// TIA Portal project "Tanques Mezcla Quimica" (V18)
// Llenado de tanques para mezcla quimica y tanque de almacenamiento

(* hardware
DEVICE "S7-1200 station_2"  S7-1200 Station
   slot 0: "Rack_0"  S7-1200 Rack  Rack  V1.0
   slot 1: "PLC_1"  CPU 1212C AC/DC/Rly  6ES7 212-1BE40-0XB0  V4.6
*)

// ===== PLC "PLC_1"  CPU 1212C AC/DC/Rly =====

VAR_GLOBAL   // PLC tag table "Default tag table_1"
   "Tag_1" AT %M1.4 : Bool;
END_VAR

VAR_GLOBAL CONSTANT   // PLC tag table "Default tag table_1"
   "None(1)" : Pip := 65535;
   "Automatic update(1)" : Pip := 0;
   "PIP 1(1)" : Pip := 1;
   "PIP 2(1)" : Pip := 2;
   "PIP 3(1)" : Pip := 3;
   "PIP 4(1)" : Pip := 4;
   "PIP OB Servo(1)" : Pip := 32768;
   "Local~MC(1)" : Hw_SubModule := 51;
   "Local~Common(1)" : Hw_SubModule := 50;
   "Local~Device(1)" : Hw_Device := 32;
   "Local~Configuration(1)" : Hw_SubModule := 33;
   "Local~Exec(1)" : Hw_SubModule := 52;
   "Local(1)" : Hw_SubModule := 49;
   "Local~PROFINET_interface_1(1)" : Hw_Interface := 64;
   "Local~PROFINET_interface_1~Port_1(1)" : Hw_Interface := 65;
   "Local~HSC_1(1)" : Hw_Hsc := 257;
   "Local~HSC_2(1)" : Hw_Hsc := 258;
   "Local~HSC_3(1)" : Hw_Hsc := 259;
   "Local~HSC_4(1)" : Hw_Hsc := 260;
   "Local~HSC_5(1)" : Hw_Hsc := 261;
   "Local~HSC_6(1)" : Hw_Hsc := 262;
   "Local~AI_2_1(1)" : Hw_SubModule := 263;
   "Local~DI_8_DQ_6_1(1)" : Hw_SubModule := 264;
   "Local~OPC_UA(1)" : Hw_SubModule := 117;
   "Local~Pulse_1(1)" : Hw_Pwm := 265;
   "Local~Pulse_2(1)" : Hw_Pwm := 266;
   "Local~Pulse_3(1)" : Hw_Pwm := 267;
   "Local~Pulse_4(1)" : Hw_Pwm := 268;
   "OB_Main(1)" : OB_PCYCLE := 1;
END_VAR

VAR_GLOBAL   // PLC tag table "IN"
   "START_MIX_PROCESS" AT %M0.0 : Bool;   // START PROCESS FOR MIX CHEMICHAL RECIPE
   "STOP_PROCESS" AT %M0.1 : Bool;   // STOP ALL THE PROCESS
   "EMERGENCY_STOP" AT %M0.2 : Bool;   // EMERGENCY STOP ALL THE PROCESS
   "TEMPERATURE_CONTROLLER" AT %M0.3 : Bool;   // TEMPERATURE CONTROLLER TANK C - CONTACT NO
   "LOW_LEVEL_TANK_C" AT %M0.4 : Bool;   // LOW LEVEL SENSOR TANK C - NO
   "LOW_LEVEL_TANK_A" AT %M0.5 : Bool;   // LOW LEVEL SENSOR TANK A - NO
   "LOW_LEVEL_TANK_B" AT %M0.6 : Bool;   // LOW LEVEL SENSOR TANK B - NO
   "HIGH_LEVEL_TANK_D" AT %M0.7 : Bool;   // HIGH LEVEL SENSOR TANK D - NO
END_VAR

VAR_GLOBAL   // PLC tag table "OUT"
   "VALVE_VA" AT %Q0.0 : Bool;   // ACTIVE VALVE A
   "VALVE_VB" AT %Q0.1 : Bool;   // ACTIVE VALVE B
   "VALVE_VD" AT %Q0.2 : Bool;   // ACTIVE VALVE D
   "PUMP" AT %Q0.3 : Bool;   // ACTIVE PUMP
   "HEATER_TANK_C" AT %Q0.4 : Bool;   // HEATER TANK C
   "VALVE_VC" AT %Q0.5 : Bool;   // ACTIVE VALVE C
END_VAR

// folder: GLOBAL VARIABLES

DATA_BLOCK "OUTPUTS"   // DB6
{ S7_Optimized_Access := 'TRUE' }
VERSION : 0.1
   VAR
      SET_RESET_PROCESS : Bool;   // START - STOP PROCESS
      OUT_TIMER_HEATER : Bool;   // OUTPUT TIMER HEATER
      OUT_TIMER_RESET_PROCESS : Bool;   // OUTPUT TIMER FOR RESET ALL PROCESS AUTO
   END_VAR
BEGIN
END_DATA_BLOCK

// folder: System blocks/Program resources

DATA_BLOCK "TIMER_DOSIFICATION_VALVE_A"   // DB1
{ S7_Optimized_Access := 'TRUE' }
AUTHOR : Simatic
FAMILY : IEC
NAME : IEC_TMR
VERSION : 1.0
// stored: InstanceOfName IEC_TIMER
"IEC_TIMER"
BEGIN
END_DATA_BLOCK

DATA_BLOCK "TIMER_DOSIFICATION_VALVE_B"   // DB2
{ S7_Optimized_Access := 'TRUE' }
AUTHOR : Simatic
FAMILY : IEC
NAME : IEC_TMR
VERSION : 1.0
// stored: InstanceOfName IEC_TIMER
"IEC_TIMER"
BEGIN
END_DATA_BLOCK

DATA_BLOCK "TIMER_HEATER_TANK_C"   // DB5
{ S7_Optimized_Access := 'TRUE' }
AUTHOR : Simatic
FAMILY : IEC
NAME : IEC_TMR
VERSION : 1.0
// stored: InstanceOfName IEC_TIMER
"IEC_TIMER"
BEGIN
END_DATA_BLOCK

DATA_BLOCK "TIMER_RESET_PROCESS"   // DB7
{ S7_Optimized_Access := 'TRUE' }
AUTHOR : Simatic
FAMILY : IEC
NAME : IEC_TMR
VERSION : 1.0
// stored: InstanceOfName IEC_TIMER
"IEC_TIMER"
BEGIN
END_DATA_BLOCK

// folder: TIMERS VALVE A-B

DATA_BLOCK "TIMERS_IN_OUT"   // DB3
{ S7_Optimized_Access := 'TRUE' }
VERSION : 0.1
   VAR
      OUT_TIMER_VA : Bool;   // OUTPUT TIMER VALVE A
      OUT_TIMER_VB : Bool;   // OUTPUT TIMER VALVE B
   END_VAR
BEGIN
END_DATA_BLOCK

// folder: (top level)

FUNCTION "START_STOP_PROCESS" : Void   // FC1, LAD
TITLE = SET - RESET PROCESS
{ S7_Optimized_Access := 'TRUE' }
VERSION : 0.1
// SET PROCESS
BEGIN

REGION Network 1: START PROCESS
   // SET PROCESS
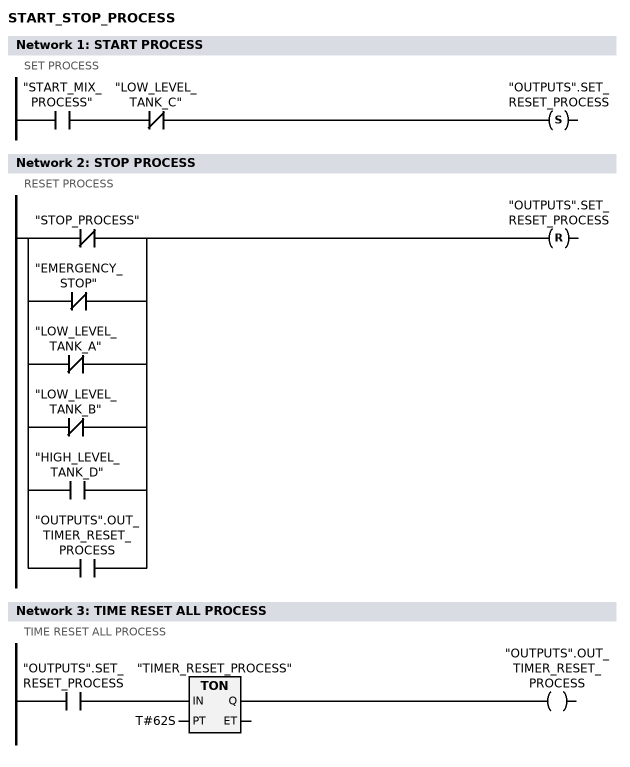
   RUNG wire#powerrail
      Contact( "START_MIX_PROCESS" )
      I_Contact( "LOW_LEVEL_TANK_C" )
      S_Coil( "OUTPUTS".SET_RESET_PROCESS )
   END_RUNG
   // the same network as SCL:
   IF "START_MIX_PROCESS" AND NOT "LOW_LEVEL_TANK_C" THEN "OUTPUTS".SET_RESET_PROCESS := TRUE; END_IF;
END_REGION

REGION Network 2: STOP PROCESS
   // RESET PROCESS
   RUNG wire#powerrail
      I_Contact( "STOP_PROCESS" )
      wire#w1
      R_Coil( "OUTPUTS".SET_RESET_PROCESS )
   END_RUNG
   RUNG wire#powerrail
      I_Contact( "EMERGENCY_STOP" )
   END_RUNG wire#w1
   RUNG wire#powerrail
      I_Contact( "LOW_LEVEL_TANK_A" )
   END_RUNG wire#w1
   RUNG wire#powerrail
      I_Contact( "LOW_LEVEL_TANK_B" )
   END_RUNG wire#w1
   RUNG wire#powerrail
      Contact( "HIGH_LEVEL_TANK_D" )
   END_RUNG wire#w1
   RUNG wire#powerrail
      Contact( "OUTPUTS".OUT_TIMER_RESET_PROCESS )
   END_RUNG wire#w1
   // the same network as SCL:
   IF NOT "STOP_PROCESS" OR NOT "EMERGENCY_STOP" OR NOT "LOW_LEVEL_TANK_A" OR NOT "LOW_LEVEL_TANK_B" OR "HIGH_LEVEL_TANK_D" OR "OUTPUTS".OUT_TIMER_RESET_PROCESS THEN
       "OUTPUTS".SET_RESET_PROCESS := FALSE;
   END_IF;
END_REGION

REGION Network 3: TIME RESET ALL PROCESS
   // TIME RESET ALL PROCESS
   "TIMER_RESET_PROCESS".TON(IN := "OUTPUTS".SET_RESET_PROCESS, PT := T#62S);
   "OUTPUTS".OUT_TIMER_RESET_PROCESS := "TIMER_RESET_PROCESS".Q;
END_REGION
END_FUNCTION

ORGANIZATION_BLOCK "Main"   // OB1, LAD, ProgramCycle
TITLE = "Main Program Sweep (Cycle)"
{ S7_Optimized_Access := 'TRUE' }
VERSION : 0.1
   VAR_INPUT
      Initial_Call : Bool;   // Initial call of this OB
      Remanence : Bool;   // =True, if remanent data are available
   END_VAR
BEGIN
END_ORGANIZATION_BLOCK

ORGANIZATION_BLOCK "Main_1"   // OB123, LAD, ProgramCycle
TITLE = "Main Program Sweep (Cycle)"
{ S7_Optimized_Access := 'TRUE' }
VERSION : 0.1
// ALL PROGRAM BLOCKS
   VAR_INPUT
      Initial_Call : Bool;   // Initial call of this OB
      Remanence : Bool;   // =True, if remanent data are available
   END_VAR
BEGIN

REGION Network 1: BLOCK SET - RESET PROCESS
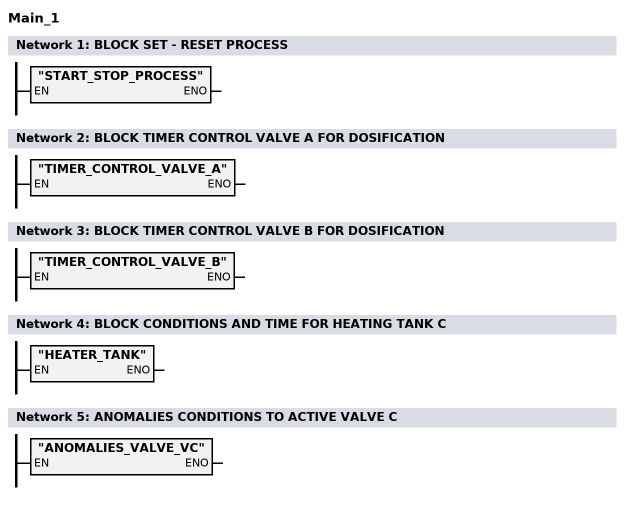
   RUNG wire#powerrail
      "START_STOP_PROCESS"()
   END_RUNG
   // the same network as SCL:
   "START_STOP_PROCESS"();
END_REGION

REGION Network 2: BLOCK TIMER CONTROL VALVE A FOR DOSIFICATION
   RUNG wire#powerrail
      "TIMER_CONTROL_VALVE_A"()
   END_RUNG
   // the same network as SCL:
   "TIMER_CONTROL_VALVE_A"();
END_REGION

REGION Network 3: BLOCK TIMER CONTROL VALVE B FOR DOSIFICATION
   RUNG wire#powerrail
      "TIMER_CONTROL_VALVE_B"()
   END_RUNG
   // the same network as SCL:
   "TIMER_CONTROL_VALVE_B"();
END_REGION

REGION Network 4: BLOCK CONDITIONS AND TIME FOR HEATING TANK C
   RUNG wire#powerrail
      "HEATER_TANK"()
   END_RUNG
   // the same network as SCL:
   "HEATER_TANK"();
END_REGION

REGION Network 5: ANOMALIES CONDITIONS TO ACTIVE VALVE C
   RUNG wire#powerrail
      "ANOMALIES_VALVE_VC"()
   END_RUNG
   // the same network as SCL:
   "ANOMALIES_VALVE_VC"();
END_REGION
END_ORGANIZATION_BLOCK

// folder: ANOMALIES CONDITIONS

FUNCTION "ANOMALIES_VALVE_VC" : Void   // FC5, LAD
TITLE = ANOMALIES TO ACTIVE VALVE C
{ S7_Optimized_Access := 'TRUE' }
VERSION : 0.1
// ANOMALIES CONDITIONS TO ACTIVE VALVE FOR DISCHARGE TANK C
BEGIN

REGION Network 1: ACTIVE VALVE C
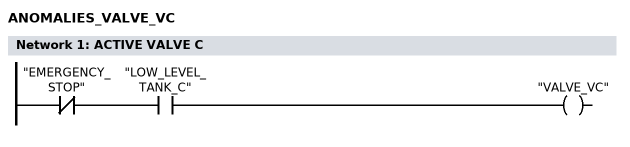
   RUNG wire#powerrail
      I_Contact( "EMERGENCY_STOP" )
      Contact( "LOW_LEVEL_TANK_C" )
      Coil( "VALVE_VC" )
   END_RUNG
   // the same network as SCL:
   "VALVE_VC" := NOT "EMERGENCY_STOP" AND "LOW_LEVEL_TANK_C";
END_REGION
END_FUNCTION

// folder: HEATER TANK C

FUNCTION "HEATER_TANK" : Void   // FC2, LAD
TITLE = START - STOP PROCESS OF HEATING, ACTIVE VALVE D AND PUMP
{ S7_Optimized_Access := 'TRUE' }
VERSION : 0.1
// CONDITIONS TO ACTIVE HEATER TANK C, CONDITIONS TO SET - RESET PUMP AND VALVE D
BEGIN

REGION Network 1: HEATER TANK C
   // CONDITIONS TO HEATING TANK C
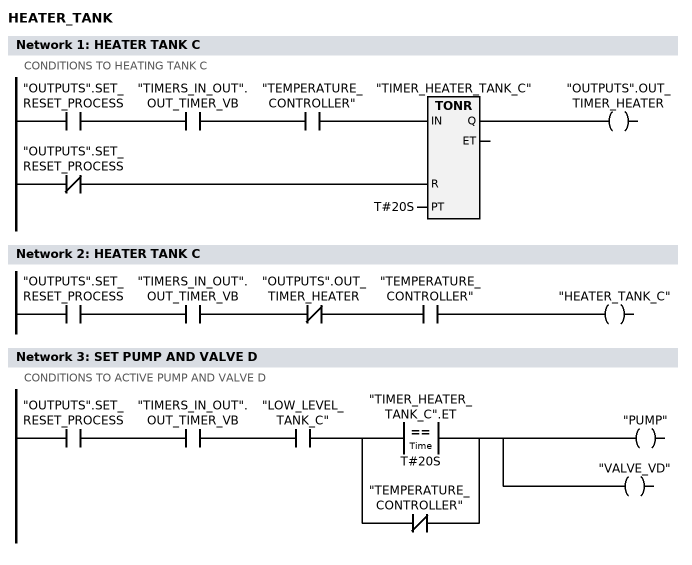
   "TIMER_HEATER_TANK_C".TONR(IN := "OUTPUTS".SET_RESET_PROCESS AND "TIMERS_IN_OUT".OUT_TIMER_VB AND "TEMPERATURE_CONTROLLER",
                           R := NOT "OUTPUTS".SET_RESET_PROCESS,
                           PT := T#20S);
   "OUTPUTS".OUT_TIMER_HEATER := "TIMER_HEATER_TANK_C".Q;
END_REGION

REGION Network 2: HEATER TANK C
   RUNG wire#powerrail
      Contact( "OUTPUTS".SET_RESET_PROCESS )
      Contact( "TIMERS_IN_OUT".OUT_TIMER_VB )
      I_Contact( "OUTPUTS".OUT_TIMER_HEATER )
      Contact( "TEMPERATURE_CONTROLLER" )
      Coil( "HEATER_TANK_C" )
   END_RUNG
   // the same network as SCL:
   "HEATER_TANK_C" := "OUTPUTS".SET_RESET_PROCESS AND "TIMERS_IN_OUT".OUT_TIMER_VB AND NOT "OUTPUTS".OUT_TIMER_HEATER AND "TEMPERATURE_CONTROLLER";
END_REGION

REGION Network 3: SET PUMP AND VALVE D
   // CONDITIONS TO ACTIVE PUMP AND VALVE D
   RUNG wire#powerrail
      Contact( "OUTPUTS".SET_RESET_PROCESS )
      Contact( "TIMERS_IN_OUT".OUT_TIMER_VB )
      Contact( "LOW_LEVEL_TANK_C" )
      wire#w1
      { S7_Templates := "SrcType := Time" } EQ_Contact(in1 := "TIMER_HEATER_TANK_C".ET, in2 := T#20S)
      wire#w2
      Coil( "PUMP" )
   END_RUNG
   RUNG wire#w1
      I_Contact( "TEMPERATURE_CONTROLLER" )
   END_RUNG wire#w2
   RUNG wire#w2
      Coil( "VALVE_VD" )
   END_RUNG
   // the same network as SCL:
   "PUMP" := "OUTPUTS".SET_RESET_PROCESS AND "TIMERS_IN_OUT".OUT_TIMER_VB AND "LOW_LEVEL_TANK_C" AND (("TIMER_HEATER_TANK_C".ET = T#20S) OR NOT "TEMPERATURE_CONTROLLER");
   "VALVE_VD" := "PUMP";
END_REGION
END_FUNCTION

// folder: TIMERS VALVE A-B

FUNCTION "TIMER_CONTROL_VALVE_A" : Void   // FC3, LAD
TITLE = DOSIFICATION CONTROL VALVE A
{ S7_Optimized_Access := 'TRUE' }
VERSION : 0.1
// TIMER AND CONDITIONS TO ACTIVE VALVE A
BEGIN

REGION Network 1: TIME CONTROL VALVE A
   // TIMER TO ACTIVE VALVE A
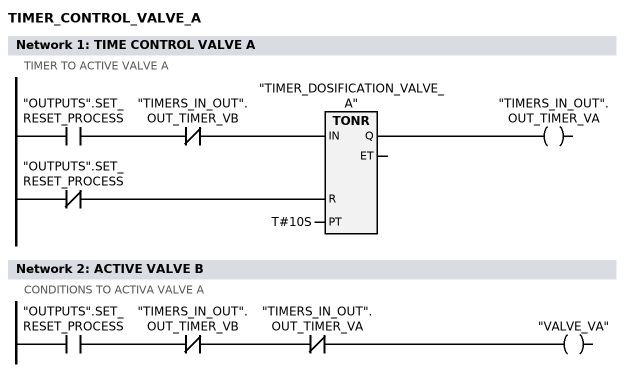
   "TIMER_DOSIFICATION_VALVE_A".TONR(IN := "OUTPUTS".SET_RESET_PROCESS AND NOT "TIMERS_IN_OUT".OUT_TIMER_VB,
                           R := NOT "OUTPUTS".SET_RESET_PROCESS,
                           PT := T#10S);
   "TIMERS_IN_OUT".OUT_TIMER_VA := "TIMER_DOSIFICATION_VALVE_A".Q;
END_REGION

REGION Network 2: ACTIVE VALVE B
   // CONDITIONS TO ACTIVA VALVE A
   RUNG wire#powerrail
      Contact( "OUTPUTS".SET_RESET_PROCESS )
      I_Contact( "TIMERS_IN_OUT".OUT_TIMER_VB )
      I_Contact( "TIMERS_IN_OUT".OUT_TIMER_VA )
      Coil( "VALVE_VA" )
   END_RUNG
   // the same network as SCL:
   "VALVE_VA" := "OUTPUTS".SET_RESET_PROCESS AND NOT "TIMERS_IN_OUT".OUT_TIMER_VB AND NOT "TIMERS_IN_OUT".OUT_TIMER_VA;
END_REGION
END_FUNCTION

FUNCTION "TIMER_CONTROL_VALVE_B" : Void   // FC4, LAD
TITLE = DOSIFICATION CONTROL VALVE B
{ S7_Optimized_Access := 'TRUE' }
VERSION : 0.1
// TIMER AND CONDICTIONS TO ACTIVE VALVE B
BEGIN

REGION Network 1: TIMER CONTROL VALVE B
   // TIMER ACTIVE VALVE B
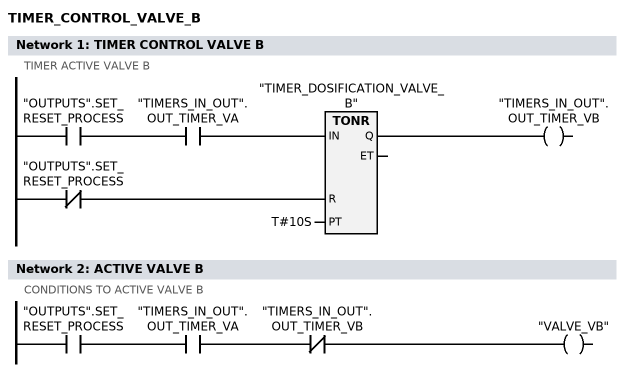
   "TIMER_DOSIFICATION_VALVE_B".TONR(IN := "OUTPUTS".SET_RESET_PROCESS AND "TIMERS_IN_OUT".OUT_TIMER_VA,
                           R := NOT "OUTPUTS".SET_RESET_PROCESS,
                           PT := T#10S);
   "TIMERS_IN_OUT".OUT_TIMER_VB := "TIMER_DOSIFICATION_VALVE_B".Q;
END_REGION

REGION Network 2: ACTIVE VALVE B
   // CONDITIONS TO ACTIVE VALVE B
   RUNG wire#powerrail
      Contact( "OUTPUTS".SET_RESET_PROCESS )
      Contact( "TIMERS_IN_OUT".OUT_TIMER_VA )
      I_Contact( "TIMERS_IN_OUT".OUT_TIMER_VB )
      Coil( "VALVE_VB" )
   END_RUNG
   // the same network as SCL:
   "VALVE_VB" := "OUTPUTS".SET_RESET_PROCESS AND "TIMERS_IN_OUT".OUT_TIMER_VA AND NOT "TIMERS_IN_OUT".OUT_TIMER_VB;
END_REGION
END_FUNCTION